(* Schneider Machine Expert - Basic project prg_control+COUNTER+RTC, file version 2.7.0.0 *)
(* ProjectInformations: Name=New project *)

HARDWARE
  Cpu 0: TM221M16R/G
  EthernetConfiguration: NetworkName=M221, IpAllocationMode=FixedAddress, IpAddress=0.0.0.0, SubnetMask=0.0.0.0
  SerialLineConfiguration: Baud=Baud19200, Parity=ParityEven, DataBits=DataBits8, StopBits=StopBits1, PhysicalMedium=PhysicalMediumRs485, TransmissionMode=TransmissionModeModbusRtu, SlaveId=1, Addressing=SlaveAddressing
  MastTask: UsePeriodScanMode=false, PeriodScan=100
  FastTask: Period=255
  CpuBehavior: StartingMode=StartAsPreviousState, AutoSaveRamOnEeprom=true, WatchdogPeriod=250

SYMBOLS  (address, symbol, comment, settings)
  %RTC0.DAY INST_RTC_DAY
  %RTC0.MONTH INST_RTC_MONTH
  %RTC0.YEAR INST_RTC_YEAR
  %RTC0.HOURS INST_RTC_HOUR
  %RTC0.MINUTES INST_RTC_MINUTE
  %RTC0.SECONDS INST_RTC_SECONDS
  %RTC0.DAYOFWEEK INST_RTC_DAYOFWEEK
  %M0       AUX_MOTOR  "Motor auxilarry"
  %M1       AUX_MACHINE  "AUX MACHINE ON"
  %M10      M_START  "M_aux_Start"
  %M11      M_STOP  "M_aux_Stop"
  %M12      M_SENSOR  "M_aux_Sensor"
  %M20      CMD_CONTROL_RESET
  %M21      IND_CONTROL_REACHED
  %M80      PET_RTC_ENABLE
  %M81      PET_RTC_READ
  %M82      PET_RTC_WRITE
  %M83      IND_RTC_DONE
  %M84      IND_RTC_ERROR
  %M90      IND_ALARM
  %M100     PET_ACK
  %M101     ALARM_01
  %M102     ALARM_02
  %MW0      IND_MOTOR_COUNTER
  %MW2      AUX_RTC_ACTUAL_TOTAL_MM
  %MW3      AUX_MACHINE_ON_TOTAL_MM
  %MW4      AUX_MACHINE_OFF_TOTAL_MM
  %MW11     CFG_COUNTER_MOTOR
  %MW12     CFG_MACHINE_ON_HH
  %MW13     CFG_MACHINE_ON_MM
  %MW14     CFG_MACHINE_OFF_HH
  %MW15     CFG_MACHINE_OFF_MM
  %MW20     IND_MOTOR_TIME
  %MW30     CFG_TIMER_MOTOR
  %MW42     IND_RTC_ACTUAL_DAY
  %MW43     IND_RTC_ACTUAL_MONTH
  %MW44     IND_RTC_ACTUAL_YEAR
  %MW45     IND_RTC_ACTUAL_HH
  %MW46     IND_RTC_ACTUAL_MM
  %MW47     IND_RTC_ACTUAL_SS
  %MW48     IND_ACTUAL_DAYOFWEEK
  %TM0      TIMER_MOTOR_ON  [Preset=5, Base=OneSecond]
  %C0         [Preset=5]
  %I0.0     I_START  "start process"
  %I0.1     I_STOP  "stop process"
  %I0.5     I_SENSOR  "detecting"
  %Q0.0     Q_MOTOR  "Motor"
  %Q0.1     Q_MACHINE_ON
  %Q0.3     Q_MACHINE_DISABLED

POU PRG RTC
  (* SectionNumber=1 *)

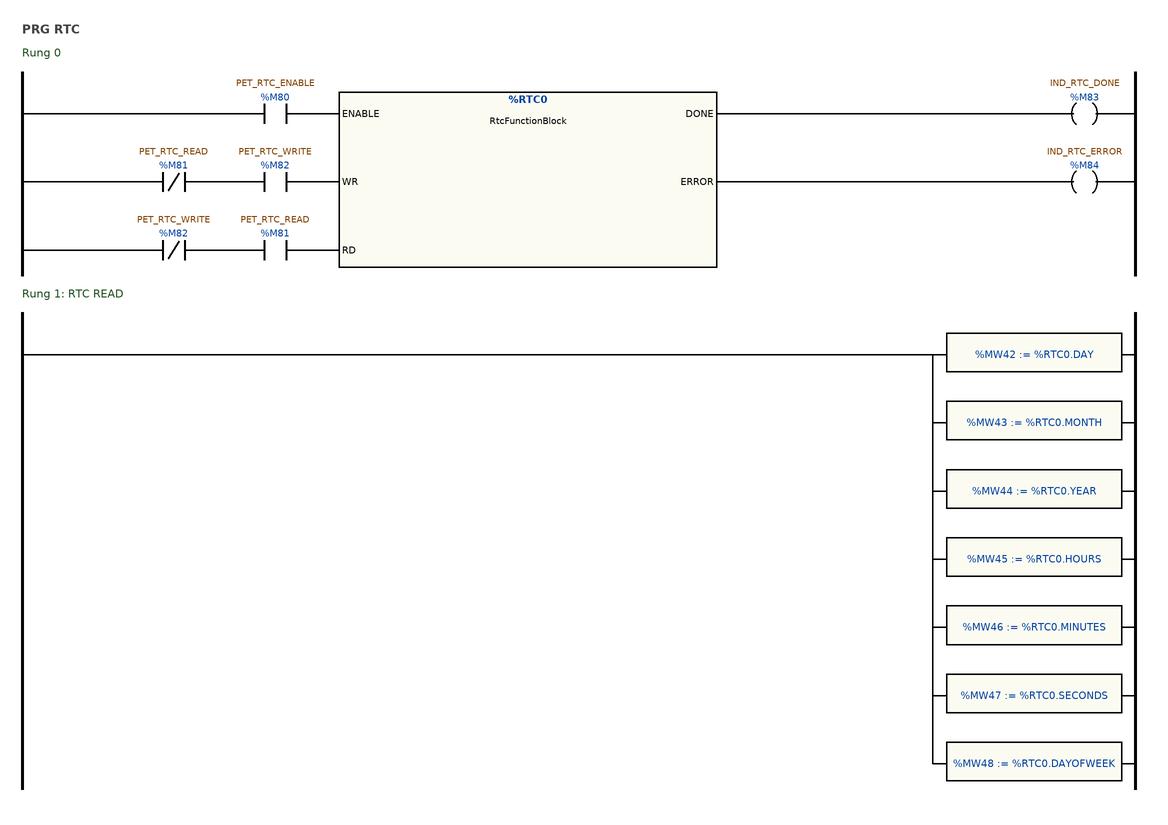

// Rung 0
  BLK %RTC0
  LD %M80                 (* PET_RTC_ENABLE *)
  ENABLE
  LDN %M81                (* PET_RTC_READ *)
  AND %M82                (* PET_RTC_WRITE *)
  WR
  LDN %M82                (* PET_RTC_WRITE *)
  AND %M81                (* PET_RTC_READ *)
  RD
  OUT_BLK
  LD DONE
  ST %M83                 (* IND_RTC_DONE *)
  LD ERROR
  ST %M84                 (* IND_RTC_ERROR *)
  END_BLK
  // as ST:
  //   %RTC0(ENABLE := PET_RTC_ENABLE, WR := NOT PET_RTC_READ AND PET_RTC_WRITE, RD := NOT PET_RTC_WRITE AND PET_RTC_READ);
  //   IND_RTC_DONE := %RTC0.DONE;
  //   IND_RTC_ERROR := %RTC0.ERROR;

// Rung 1: RTC READ
  LD 1
  [ %MW42 := %RTC0.DAY ]  (* IND_RTC_ACTUAL_DAY *)
  [ %MW43 := %RTC0.MONTH ](* IND_RTC_ACTUAL_MONTH *)
  [ %MW44 := %RTC0.YEAR ] (* IND_RTC_ACTUAL_YEAR *)
  [ %MW45 := %RTC0.HOURS ](* IND_RTC_ACTUAL_HH *)
  [ %MW46 := %RTC0.MINUTES ](* IND_RTC_ACTUAL_MM *)
  [ %MW47 := %RTC0.SECONDS ](* IND_RTC_ACTUAL_SS *)
  [ %MW48 := %RTC0.DAYOFWEEK ](* IND_ACTUAL_DAYOFWEEK *)
  // as ST:
  //   IND_RTC_ACTUAL_DAY := %RTC0.DAY;
  //   IND_RTC_ACTUAL_MONTH := %RTC0.MONTH;
  //   IND_RTC_ACTUAL_YEAR := %RTC0.YEAR;
  //   IND_RTC_ACTUAL_HH := %RTC0.HOURS;
  //   IND_RTC_ACTUAL_MM := %RTC0.MINUTES;
  //   IND_RTC_ACTUAL_SS := %RTC0.SECONDS;
  //   IND_ACTUAL_DAYOFWEEK := %RTC0.DAYOFWEEK;

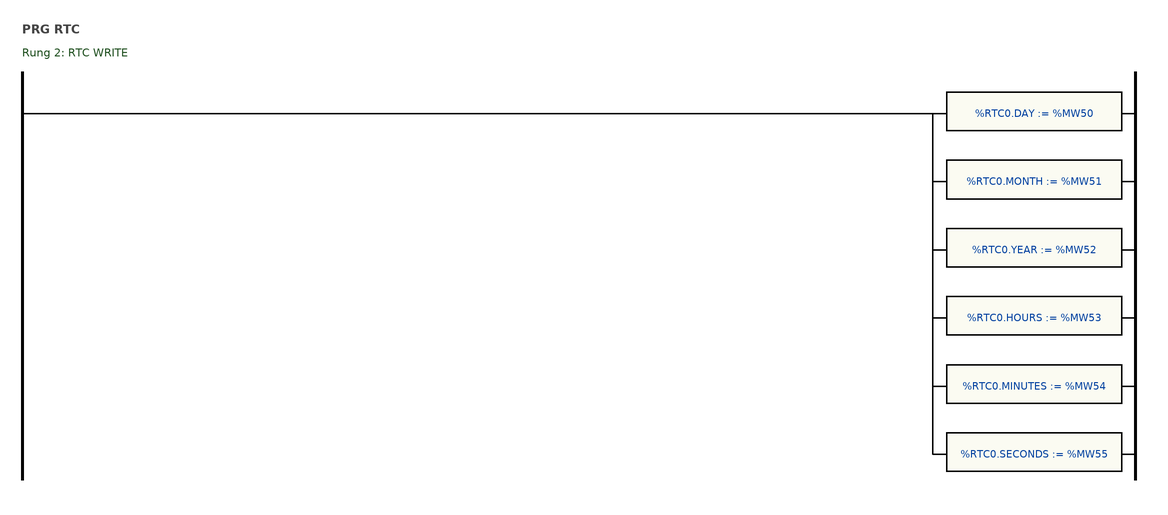

// Rung 2: RTC WRITE
  LD 1
  [ %RTC0.DAY := %MW50 ]
  [ %RTC0.MONTH := %MW51 ]
  [ %RTC0.YEAR := %MW52 ]
  [ %RTC0.HOURS := %MW53 ]
  [ %RTC0.MINUTES := %MW54 ]
  [ %RTC0.SECONDS := %MW55 ]
  // as ST:
  //   %RTC0.DAY := %MW50;
  //   %RTC0.MONTH := %MW51;
  //   %RTC0.YEAR := %MW52;
  //   %RTC0.HOURS := %MW53;
  //   %RTC0.MINUTES := %MW54;
  //   %RTC0.SECONDS := %MW55;

POU PRG CONFIG
  (* SectionNumber=2 *)

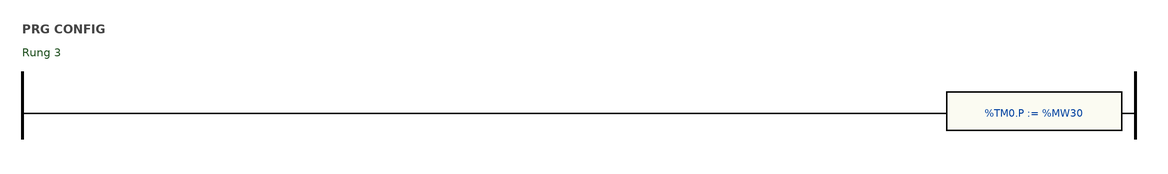

// Rung 3
  LD 1
  [ %TM0.P := %MW30 ]     (* TIMER_MOTOR_ON, CFG_TIMER_MOTOR *)
  // as ST:
  //   TIMER_MOTOR_ON.P := CFG_TIMER_MOTOR;

POU PRG INPUTS
  (* SectionNumber=3 *)

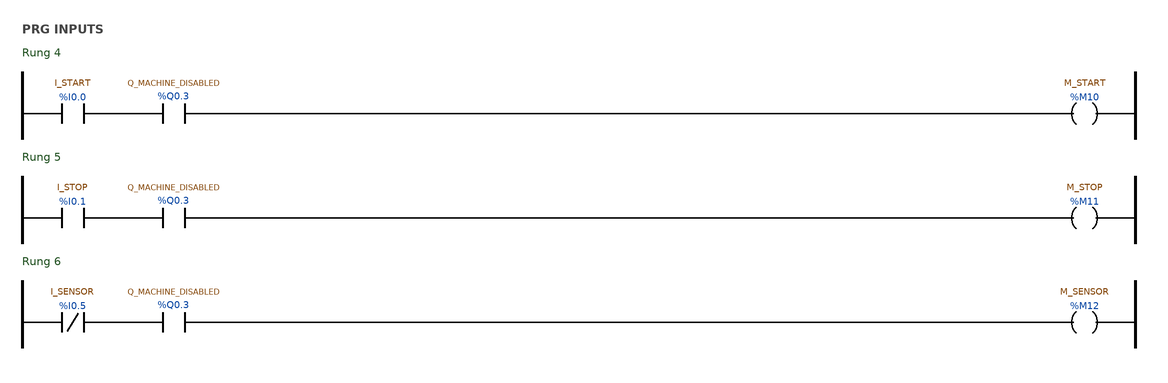

// Rung 4
  LD %I0.0                (* I_START *)
  AND %Q0.3               (* Q_MACHINE_DISABLED *)
  ST %M10                 (* M_START *)
  // as ST:
  //   M_START := I_START AND Q_MACHINE_DISABLED;

// Rung 5
  LD %I0.1                (* I_STOP *)
  AND %Q0.3               (* Q_MACHINE_DISABLED *)
  ST %M11                 (* M_STOP *)
  // as ST:
  //   M_STOP := I_STOP AND Q_MACHINE_DISABLED;

// Rung 6
  LDN %I0.5               (* I_SENSOR *)
  AND %Q0.3               (* Q_MACHINE_DISABLED *)
  ST %M12                 (* M_SENSOR *)
  // as ST:
  //   M_SENSOR := NOT I_SENSOR AND Q_MACHINE_DISABLED;

POU PRG_Control
  (* SectionNumber=4 *)

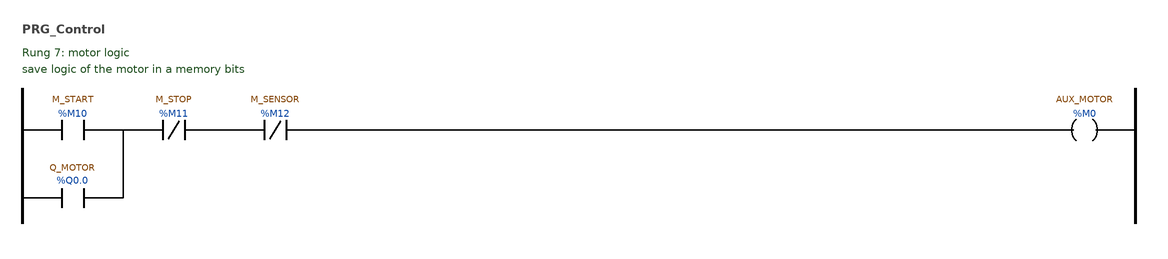

// Rung 7: motor logic
// save logic of the motor in a memory bits
  LD %M10                 (* M_START *)
  OR %Q0.0                (* Q_MOTOR *)
  ANDN %M11               (* M_STOP *)
  ANDN %M12               (* M_SENSOR *)
  ST %M0                  (* AUX_MOTOR *)
  // as ST:
  //   AUX_MOTOR := (M_START OR Q_MOTOR) AND NOT M_STOP AND NOT M_SENSOR;

POU PRG OUTPUT
  (* SectionNumber=5 *)

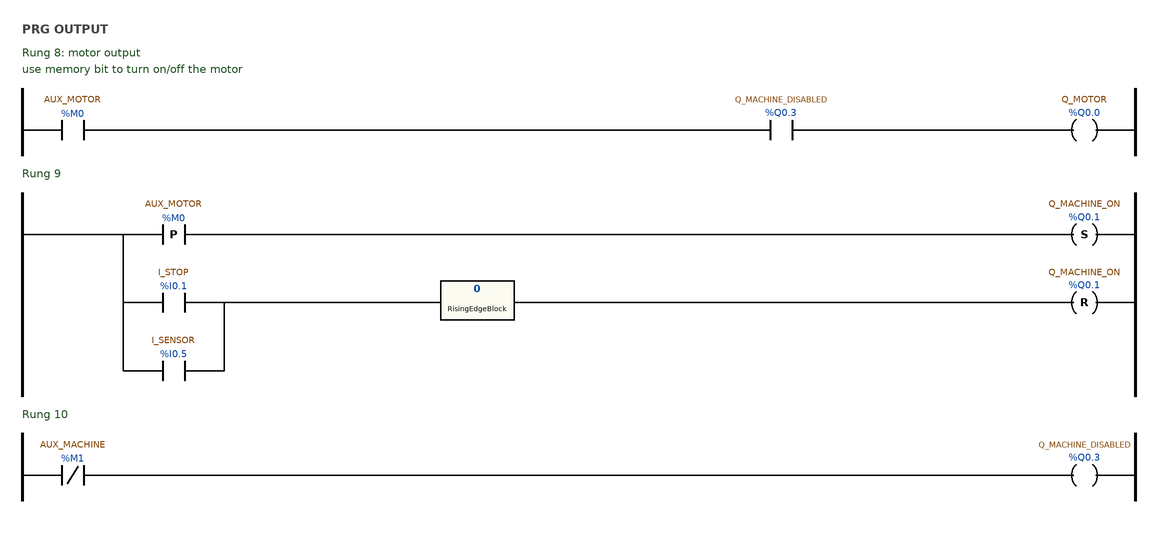

// Rung 8: motor output
// use memory bit to turn on/off the motor
  LD %M0                  (* AUX_MOTOR *)
  AND %Q0.3               (* Q_MACHINE_DISABLED *)
  ST %Q0.0                (* Q_MOTOR *)
  // as ST:
  //   Q_MOTOR := AUX_MOTOR AND Q_MACHINE_DISABLED;

// Rung 9
  LD 1
  MPS
  ANDR %M0                (* AUX_MOTOR *)
  S %Q0.1                 (* Q_MACHINE_ON *)
  MPP
  AND( %I0.1              (* I_STOP *)
  OR %I0.5                (* I_SENSOR *)
  )
  RISING0
  R %Q0.1                 (* Q_MACHINE_ON *)
  // as ST:
  //   IF RISING(AUX_MOTOR) THEN Q_MACHINE_ON := TRUE; END_IF;
  //   IF RISING(I_STOP OR I_SENSOR) THEN Q_MACHINE_ON := FALSE; END_IF;

// Rung 10
  LDN %M1                 (* AUX_MACHINE *)
  ST %Q0.3                (* Q_MACHINE_DISABLED *)
  // as ST:
  //   Q_MACHINE_DISABLED := NOT AUX_MACHINE;

POU PRG ALArm
  (* SectionNumber=6 *)

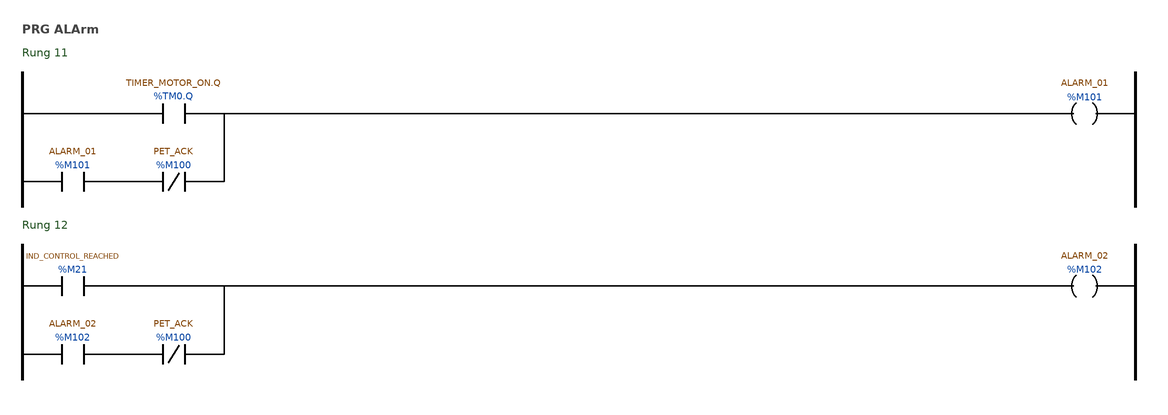

// Rung 11
  LD 1
  AND %TM0.Q              (* TIMER_MOTOR_ON *)
  OR( %M101               (* ALARM_01 *)
  ANDN %M100              (* PET_ACK *)
  )
  ST %M101                (* ALARM_01 *)
  // as ST:
  //   ALARM_01 := TIMER_MOTOR_ON.Q OR ALARM_01 AND NOT PET_ACK;

// Rung 12
  LD %M21                 (* IND_CONTROL_REACHED *)
  OR( %M102               (* ALARM_02 *)
  ANDN %M100              (* PET_ACK *)
  )
  ST %M102                (* ALARM_02 *)
  // as ST:
  //   ALARM_02 := IND_CONTROL_REACHED OR ALARM_02 AND NOT PET_ACK;

POU PRG MGMT
  (* SectionNumber=7 *)

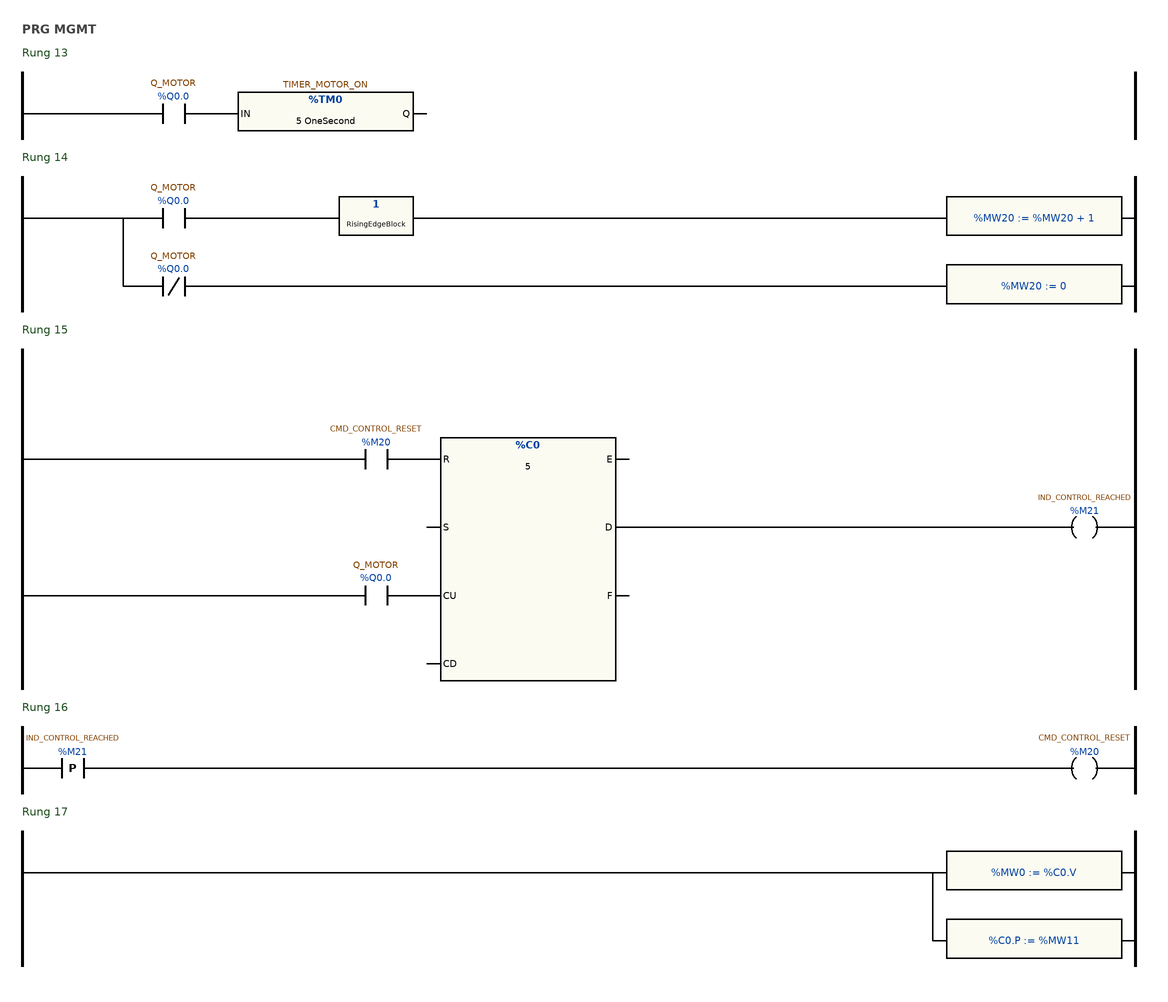

// Rung 13
  BLK %TM0                (* TIMER_MOTOR_ON *)
  LD %Q0.0                (* Q_MOTOR *)
  IN
  END_BLK
  // as ST:
  //   TIMER_MOTOR_ON(IN := Q_MOTOR);

// Rung 14
  LD 1
  MPS
  AND %Q0.0               (* Q_MOTOR *)
  RISING1
  [ %MW20 := %MW20 + 1 ]  (* IND_MOTOR_TIME, IND_MOTOR_TIME *)
  MPP
  ANDN %Q0.0              (* Q_MOTOR *)
  [ %MW20 := 0 ]          (* IND_MOTOR_TIME *)
  // as ST:
  //   IF RISING(Q_MOTOR) THEN IND_MOTOR_TIME := IND_MOTOR_TIME + 1; END_IF;
  //   IF NOT Q_MOTOR THEN IND_MOTOR_TIME := 0; END_IF;

// Rung 15
  BLK %C0
  LD %M20                 (* CMD_CONTROL_RESET *)
  R
  LD %Q0.0                (* Q_MOTOR *)
  CU
  OUT_BLK
  LD D
  ST %M21                 (* IND_CONTROL_REACHED *)
  END_BLK
  // as ST:
  //   %C0(R := CMD_CONTROL_RESET, CU := Q_MOTOR);
  //   IND_CONTROL_REACHED := %C0.D;

// Rung 16
  LDR %M21                (* IND_CONTROL_REACHED *)
  ST %M20                 (* CMD_CONTROL_RESET *)
  // as ST:
  //   CMD_CONTROL_RESET := RISING(IND_CONTROL_REACHED);

// Rung 17
  LD 1
  [ %MW0 := %C0.V ]       (* IND_MOTOR_COUNTER *)
  [ %C0.P := %MW11 ]      (* CFG_COUNTER_MOTOR *)
  // as ST:
  //   IND_MOTOR_COUNTER := %C0.V;
  //   %C0.P := CFG_COUNTER_MOTOR;

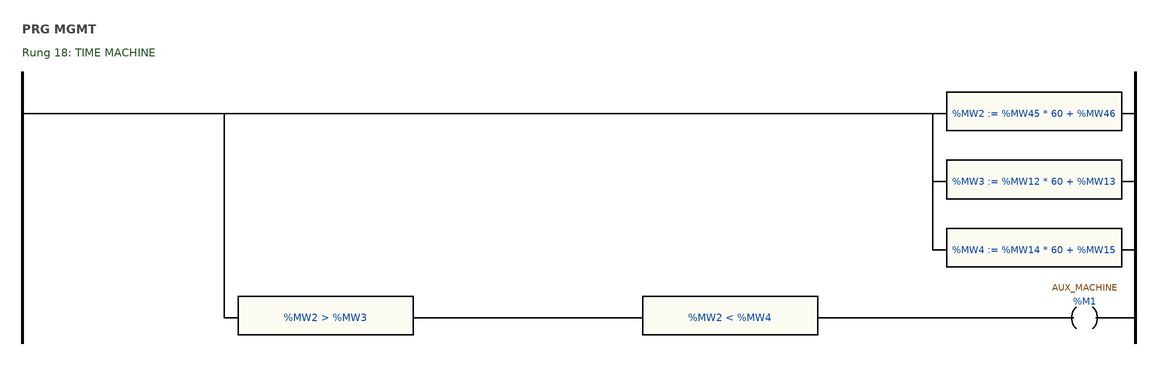

// Rung 18: TIME MACHINE
  LD 1
  MPS
  [ %MW2 := %MW45 * 60 + %MW46 ](* AUX_RTC_ACTUAL_TOTAL_MM, IND_RTC_ACTUAL_HH, IND_RTC_ACTUAL_MM *)
  [ %MW3 := %MW12 * 60 + %MW13 ](* AUX_MACHINE_ON_TOTAL_MM, CFG_MACHINE_ON_HH, CFG_MACHINE_ON_MM *)
  [ %MW4 := %MW14 * 60 + %MW15 ](* AUX_MACHINE_OFF_TOTAL_MM, CFG_MACHINE_OFF_HH, CFG_MACHINE_OFF_MM *)
  MPP
  AND [ %MW2 > %MW3 ]     (* AUX_RTC_ACTUAL_TOTAL_MM, AUX_MACHINE_ON_TOTAL_MM *)
  AND [ %MW2 < %MW4 ]     (* AUX_RTC_ACTUAL_TOTAL_MM, AUX_MACHINE_OFF_TOTAL_MM *)
  ST %M1                  (* AUX_MACHINE *)
  // as ST:
  //   AUX_RTC_ACTUAL_TOTAL_MM := IND_RTC_ACTUAL_HH * 60 + IND_RTC_ACTUAL_MM;
  //   AUX_MACHINE_ON_TOTAL_MM := CFG_MACHINE_ON_HH * 60 + CFG_MACHINE_ON_MM;
  //   AUX_MACHINE_OFF_TOTAL_MM := CFG_MACHINE_OFF_HH * 60 + CFG_MACHINE_OFF_MM;
  //   AUX_MACHINE := AUX_RTC_ACTUAL_TOTAL_MM > AUX_MACHINE_ON_TOTAL_MM AND AUX_RTC_ACTUAL_TOTAL_MM < AUX_MACHINE_OFF_TOTAL_MM;

POU PRG GRALS ALARM
  (* SectionNumber=8 *)

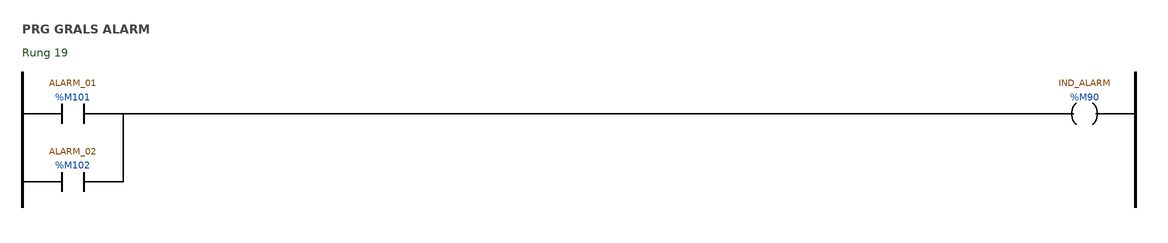

// Rung 19
  LD %M101                (* ALARM_01 *)
  OR %M102                (* ALARM_02 *)
  ST %M90                 (* IND_ALARM *)
  // as ST:
  //   IND_ALARM := ALARM_01 OR ALARM_02;
